Universal Robots PolyScope program: v2.2ross.urp

Program v2.2ross (installation=botross directory=/programs/usbdisk/APS2OsUltimosRomanticos createdIn=3.15.3.106223 lastSavedIn=3.15.3.106223 robotSerialNumber=2017357016)
Calibrated DH parameters: a=[0.000101, -0.084242, -0.391552, -0.00002, 0.000081, 0]; d=[0.089343, 205.941147, -210.196002, 4.364986, 0.094781, 0.082586]; alpha=[1.56998, -0.002024, -0.006166, 1.570936, -1.570286, 0]; deltaTheta=[0.000038, -1.371443, 1.438374, -0.066933, 0.000048, 0.000033]
BeforeStart
  Socket := socket_open("10.103.16.11",20000)
  Num_points := socket_read_ascii_float(1)
Robot Program (runOnlyOnce=false)
  Loop While (checkContinuously=false) expression=Socket≟ False
    Socket := socket_open("10.103.16.11",20000)
  Num_points := socket_read_ascii_float(1)
  N := Num_points[1]
  X := socket_read_ascii_float(N)
  Y := socket_read_ascii_float(N)
  Z := socket_read_ascii_float(N)
  SuppressedNode
    Socket := socket_close()
  count := 1
  Loop While (checkContinuously=false) expression=count≤N
    move2pose := p[X[count]/1000,Y[count]/1000,Z[count]/1000,0,0,0]
    MoveL speed 200 mm/s, acceleration 600 mm/s^2 (useActiveTCP=true) feature=Plano_BotRoss
      Waypoint Waypoint (Variable): variable=move2pose
    SuppressedNode
      Wait Sleep waitTime=0.5
    count := count+1
  SuppressedNode
    Script: socket_close()
Thread Thread_1 (runOnlyOnce=false)
  Loop While (checkContinuously=false) expression=Socket≟ False
    Socket := socket_open("10.103.16.11",20000)
  Set Undefined
  Switch
Event 
  Wait Sleep waitTime=180
Thread Thread_2 (runOnlyOnce=false)
  Socket := socket_open("10.103.16.11",20000)
Thread Thread_3 (runOnlyOnce=false)
  Socket := socket_open("10.103.16.11",20000)
